// TIA Portal project "AWL SEMAFORO" (V11)

(* hardware
DEVICE "S7300/ET200 station_1"  SIMATIC 300-Station
   slot 0: "Perfil soporte_0"  Rail  6ES7 390-1***0-0AA0
   slot 2: "PLC_1"  CPU 313C-2 DP  6ES7 313-6CF03-0AB0  V2.6
      slot 0: "Interfaz MPI_1"  MPI
      slot 1: "Interfaz DP_1"  DP
      slot 2: "DI16/DO16_1"  DI16/DO16
      slot 4: "Contaje_1"  Counter
*)

// ===== PLC "PLC_1"  CPU 313C-2 DP =====

VAR_GLOBAL   // PLC tag table "Tabla de variables estándar"
   "PULSADOR" AT %E0.0 : Bool;
   "VERDE COCHE" AT %A0.0 : Bool;
   "AMBAR COCHE" AT %A0.1 : Bool;
   "ROJO COCHE" AT %A0.2 : Bool;
   "ROJO PEATON" AT %A0.3 : Bool;
   "VERDE PEATON" AT %A0.4 : Bool;
   "Tag_1" AT %M0.0 : Bool;
   "Tag_2" AT %M0.1 : Bool;
   "Tag_3" AT %T0 : Timer;
   "Tag_4" AT %MB0 : Byte;
   "Tag_5" AT %AB0 : Byte;
   "Tag_6" AT %M0.2 : Bool;
   "Tag_7" AT %M0.3 : Bool;
   "Tag_8" AT %T1 : Timer;
   "Tag_9" AT %M0.4 : Bool;
   "Tag_10" AT %T2 : Timer;
   "Tag_11" AT %M0.5 : Bool;
   "Tag_12" AT %A0.7 : Bool;
   "Tag_13" AT %T3 : Timer;
   "Tag_14" AT %M0.6 : Bool;
   "Tag_15" AT %MB10 : Byte;
   "Tag_16" AT %M10.0 : Bool;
   "Tag_17" AT %M10.1 : Bool;
   "Tag_18" AT %M10.2 : Bool;
   "Tag_19" AT %M10.3 : Bool;
   "Tag_20" AT %M10.4 : Bool;
   "Tag_21" AT %M10.7 : Bool;
END_VAR

ORGANIZATION_BLOCK "Main"   // OB1, STL
TITLE = "Main Program Sweep (Cycle)"
{ S7_Optimized_Access := 'FALSE' }
VERSION : 0.1
   VAR_TEMP
      OB1_EV_CLASS : Byte;   // Bits 0-3 = 1 (Coming event), Bits 4-7 = 1 (Event class 1)
      OB1_SCAN_1 : Byte;   // 1 (Cold restart scan 1 of OB 1), 3 (Scan 2-n of OB 1)
      OB1_PRIORITY : Byte;   // Priority of OB Execution
      OB1_OB_NUMBR : Byte;   // 1 (Organization block 1, OB1)
      OB1_RESERVED_1 : Byte;   // Reserved for system
      OB1_RESERVED_2 : Byte;   // Reserved for system
      OB1_PREV_CYCLE : Int;   // Cycle time of previous OB1 scan (milliseconds)
      OB1_MIN_CYCLE : Int;   // Minimum cycle time of OB1 (milliseconds)
      OB1_MAX_CYCLE : Int;   // Maximum cycle time of OB1 (milliseconds)
      OB1_DATE_TIME : Date_And_Time;   // Date and time OB1 started
   END_VAR
BEGIN

REGION Network 1
         AN    "Tag_1";  // ENTRADA DIRECTA.
         FP    "Tag_2";  // FLANCO P.
         JNB   _001;
         L     B#16#9;  // VERDE COCHES - ROJO PEATONES.
         T     "Tag_15";
   _001: NOP   0;
         A     "PULSADOR";  // INICIO SECUENCIA PEATONES.
         FP    "Tag_6";
         JNB   _002;
         L     B#16#0A;  // AMBAR COCHES - ROJO PEATONES.
         T     "Tag_15";
   _002: NOP   0;
         A     "AMBAR COCHE";
         L     S5T#3S;  // PRIMERA TEMPORIZACION 3S.
         SD    "Tag_3";  // T0 A LA CONEXION.
         A     "Tag_3";  // CONTACTO TEMPORZADO T0.
         FP    "Tag_7";
         JNB   _003;
         L     B#16#0C;  // ROJO COCHES - ROJO PEATONES.
         T     "Tag_15";
   _003: NOP   0;
         A     "ROJO COCHE";
         L     S5T#3S;  // SEGUNDA TEMPORIZACION 3S.
         SD    "Tag_8";  // T1 A LA CONEXION.
         A     "Tag_8";  // CONTACTO TEMPORIZADO T1.
         FP    "Tag_9";
         JNB   _004;
         L     B#16#14;  // ROJO COCHES - VERDE PEATON .
         T     "Tag_15";
   _004: NOP   0;
         A     "VERDE PEATON";
         L     S5T#14S;  // TERCERA TEMPORIZACION 14S.
         SD    "Tag_10";  // T2 A LA CONEXION.
         A     "Tag_10";  // CONTACTO TEMPORIZADO T2.
         FP    "Tag_11";
         JNB   _005;
         L     B#16#8C;  // ROJO COCHES - ROJO PEATONES
         T     "Tag_15";
   _005: NOP   0;
         A     "Tag_21";  // AUXILIAR PARA NO CONFUNDIR LA SECUENCIA.
         L     S5T#3S;  // CUARTA TEMPORIZACION 3S.
         SD    "Tag_13";  // T3 A LA CONEXION.
         A     "Tag_13";  //CONTACO TEMPORIZADO T3.
         FP    "Tag_14";
         JNB   _006;
         L     B#16#9;
         T     "Tag_15";
   _006: NOP   0;
         A     "Tag_16";
         =     "VERDE COCHE";
         A     "Tag_17";
         =     "AMBAR COCHE";
         A     "Tag_18";
         =     "ROJO COCHE";
         A     "Tag_19";
         =     "ROJO PEATON";
         A     "Tag_20";
         =     "VERDE PEATON";
END_REGION
END_ORGANIZATION_BLOCK